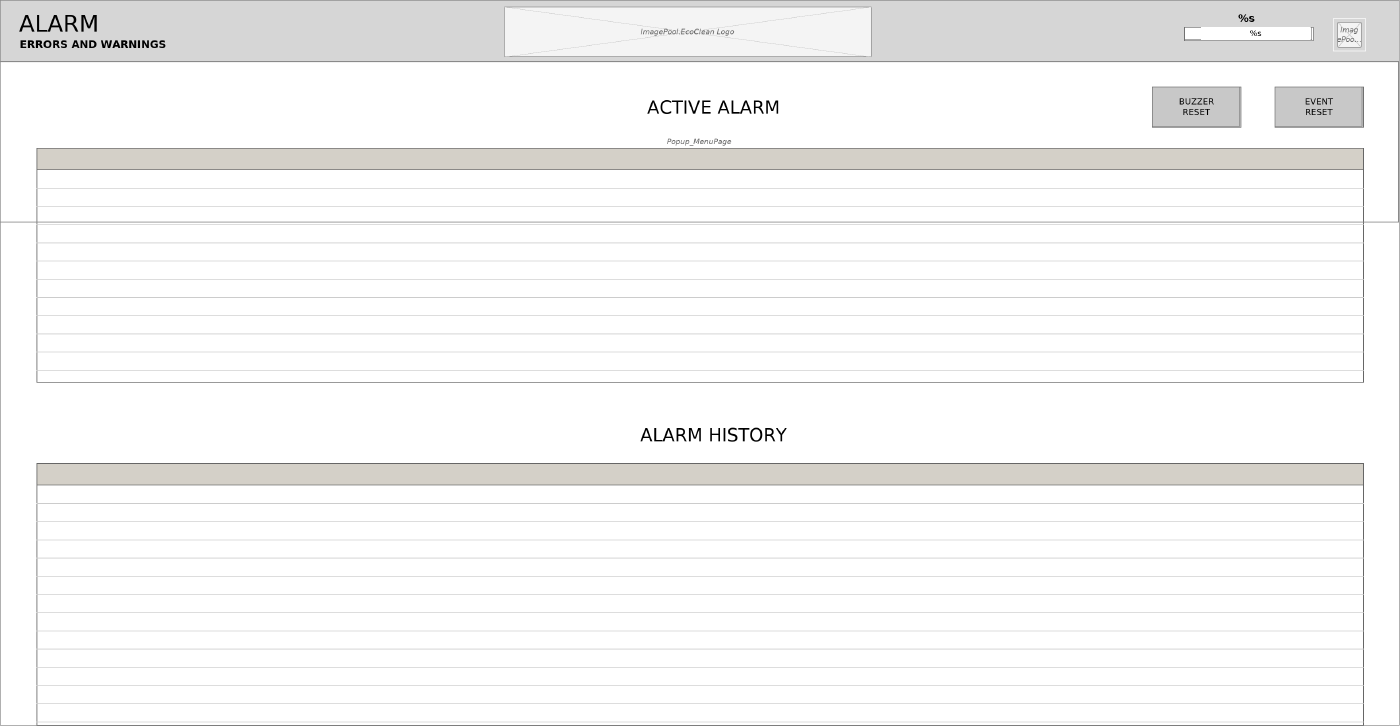
VISUALIZATION Alarm_Page  // 1920x997
    Rectangle (0,63 1920x26)
        p3528305787: HMI_Ctrl.ANIMATION3
    Rectangle (0,0 1919x85)
    Label (23,6 267x53), "ALARM"
    Label (24,49 320x24), "ERRORS AND WARNINGS"
    Group (1828,25 45x45)
        OnMouseClick: toggle HMI_Ctrl.MenuButton
        RoundedRectangle (0,0 45x45), colour toggle: HMI_Ctrl.MenuButton
        Image (6,5 33x35), image: ImagePool.Menu Button
    Rectangle (769,133 419x29), "ACTIVE ALARM"
    Rectangle (769,583 419x29), "ALARM HISTORY"
    Button (1748,119 122x56), "EVENT RESET"
        tap bEventRstPB
    Button (1580,119 122x56), "BUZZER RESET"
        tap bBuzzerRstPB
    Table (50,203 1820x322), data array: ARdsEventActiveDisplay
        p3854506369: ARdsEventActiveDisplay[INDEX].iEventID
        p1892666644: ARdsEventActiveDisplay[INDEX].sTimeAndDate_Occurred
        p338671338: ARdsEventActiveDisplay[INDEX].sEventCode
        p2170511999: ARdsEventActiveDisplay[INDEX].sEventType
        p3723444502: ARdsEventActiveDisplay[INDEX].sLocation
        p1218418051: ARdsEventActiveDisplay[INDEX].sSubLocation
        p746581629: ARdsEventActiveDisplay[INDEX].sDescription
        p3104783080: ARdsEventActiveDisplay[INDEX].sCaused
        p2501879983: ARdsEventActiveDisplay[INDEX].sRemedy
        p2232123230: EVENT ID
        p1791247317: ARdsEventActiveDisplay[INDEX].sEventType_C
    Table (50,636 1820x361), data array: ARdsEventHistoryDisplay
        p3854506369: ARdsEventHistoryDisplay[INDEX].iEventID
        p7306298: ARdsEventHistoryDisplay[INDEX].sCaused
        p1933151965: ARdsEventHistoryDisplay[INDEX].sRemedy
        p1892666644: ARdsEventHistoryDisplay[INDEX].sEventCode
        p511219082: EVENT ID
        p338671338: ARdsEventHistoryDisplay[INDEX].sTimeAndDate_Occurred
        p4092479075: ARdsEventHistoryDisplay[INDEX].sTimeAndDate_Acknowledged
        p2237128397: ARdsEventHistoryDisplay[INDEX].sEventType
        p505689113: ARdsEventHistoryDisplay[INDEX].sLocation
        p1757482276: ARdsEventHistoryDisplay[INDEX].sSubLocation
        p3104783080: ARdsEventHistoryDisplay[INDEX].sDescription
        p2501879983: ARdsEventHistoryDisplay[INDEX].sTimeAndDate_Recovered
    Frame (0,84 1918x221), invisible if: HMI_Ctrl.CloseMenuButton
        shows Popup_MenuPage()
    Image (691,9 504x69), image: ImagePool.EcoClean Logo
    Group (1621,14 180x42)
        Rectangle (0,0 177x22), "%s", text variable: DSLocalSystemTimeML.sCurrentDT24Hr_General
        Button (3,23 177x19), image: VisuSymbols.Symbols.AddUser
        Rectangle (26,23 150x18), "%s", text variable: fbHmiTF1800_UserlevelManagement.dsHmiUserStatus_Active.sLoginName
END_VISUALIZATION

(* stored: Version 1.1.0.1, ProductVersion 3.1.4024.12
   Visu Alarm_Page: Id {d6b14665-0f6d-47bf-8a90-77e885e9a03a} *)
